FUNCTION F_Bel_Daten_Lesen : BOOL
VAR_IN_OUT
	Zustand	: ST_PU_Zustand;
END_VAR
VAR_INPUT
	StatusModul1	: DWORD;
	StatusModul2	: DWORD;
END_VAR
VAR
END_VAR

Zustand.Stoerung_Code.0 	:= StatusModul1.1;

END_FUNCTION

(* stored: Version 1.1.0.1, ProductVersion 3.1.4024.10
   POU F_Bel_Daten_Lesen: Id {74359aab-bc83-4bf2-9b5b-de8991304bba}, SpecialFunc None *)
